(* Logix 5000 project; controller Drives_Line1 1756-L72 rev 20.13; software revision 20.04; part 4 of 21 *)
(* tags used below, declared in another part *)
   EOC_ToCoilerStep : DINT;
   Exit_PosPv_Winder : REAL;
   zMaxSpdExitNotSync : REAL;
   Exit_Accu : UDT_Exit_Accu;
   Exit_PosSp_ToWinder : DINT;
   ExitCmd : UDT_Commands_Zone;
   ExitConfig : UDT_Config_Zone;
   ExitCtrl : UDT_Control_Zone;
   ExitFdbks : UDT_Feedbacks_Zone;
   ExitSetpoints : UDT_Setpoints_Zone;
   ExitStat : UDT_Status_Zone;
   In_Commands : UDT_Commands;
   In_Config : UDT_Config;
   In_Setpoints : UDT_Setpoints;
   LineCmd : UDT_Commands_Line;
   LineStat : UDT_Status_Line;
   Out_Feedbacks : UDT_Fdbks;
   Out_Status : UDT_Status;
   TestConfig_Exit : UDT_Config_Zone;
   Unwinder_1 : UDT_Unwinder;
   Winder : UDT_Winder;
   Winder_FB_Counts_Diff : DINT;
   Winder_FB_Counts_mm : DINT;
   Winder_FB_Update_Valid : BOOL;
   zConfigFromMaster : BOOL;
   zExit_Dist_ShearToWinder : DINT;
   zWinderDiamFullTrq : REAL;
(* P02_Exit_Zone, continued *)

ROUTINE R03_EOC_ToCoiler   (* ladder *)
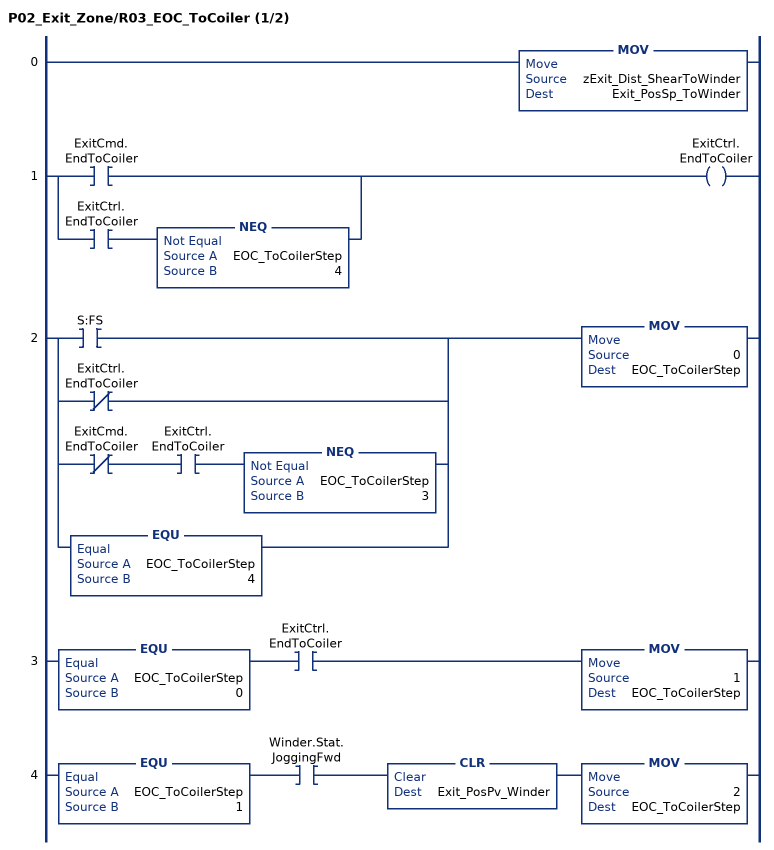
   0: MOV(zExit_Dist_ShearToWinder,Exit_PosSp_ToWinder);
   1: [XIC(ExitCmd.EndToCoiler) ,XIC(ExitCtrl.EndToCoiler) NEQ(EOC_ToCoilerStep,4) ]OTE(ExitCtrl.EndToCoiler);
   2: [XIC(S:FS) ,XIO(ExitCtrl.EndToCoiler) ,XIO(ExitCmd.EndToCoiler) XIC(ExitCtrl.EndToCoiler) NEQ(EOC_ToCoilerStep,3) ,EQU(EOC_ToCoilerStep,4) ]MOV(0,EOC_ToCoilerStep);
   3: EQU(EOC_ToCoilerStep,0)XIC(ExitCtrl.EndToCoiler)MOV(1,EOC_ToCoilerStep);
   4: EQU(EOC_ToCoilerStep,1)XIC(Winder.Stat.JoggingFwd)CLR(Exit_PosPv_Winder)MOV(2,EOC_ToCoilerStep);
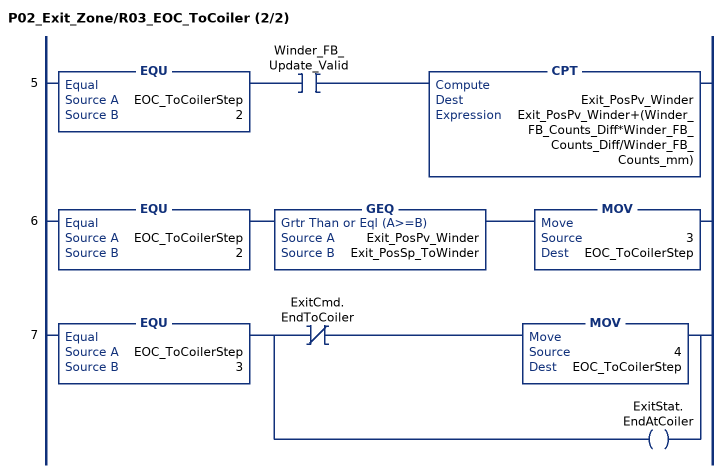
   5: EQU(EOC_ToCoilerStep,2)XIC(Winder_FB_Update_Valid)CPT(Exit_PosPv_Winder,Exit_PosPv_Winder+(Winder_FB_Counts_Diff*Winder_FB_Counts_Diff/Winder_FB_Counts_mm));
   6: EQU(EOC_ToCoilerStep,2)GEQ(Exit_PosPv_Winder,Exit_PosSp_ToWinder)MOV(3,EOC_ToCoilerStep);
   7: EQU(EOC_ToCoilerStep,3)[XIO(ExitCmd.EndToCoiler) MOV(4,EOC_ToCoilerStep) ,OTE(ExitStat.EndAtCoiler) ];
END_ROUTINE

ROUTINE R05_Control   (* ladder *)
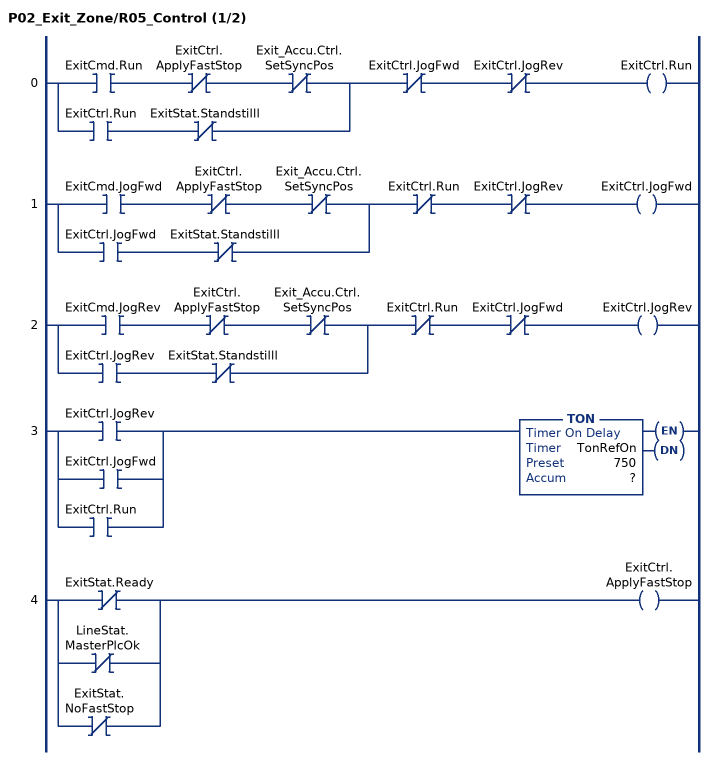
   0: [XIC(ExitCmd.Run) XIO(ExitCtrl.ApplyFastStop) XIO(Exit_Accu.Ctrl.SetSyncPos) ,XIC(ExitCtrl.Run) XIO(ExitStat.Standstilll) ]XIO(ExitCtrl.JogFwd)XIO(ExitCtrl.JogRev)OTE(ExitCtrl.Run);
   1: [XIC(ExitCmd.JogFwd) XIO(ExitCtrl.ApplyFastStop) XIO(Exit_Accu.Ctrl.SetSyncPos) ,XIC(ExitCtrl.JogFwd) XIO(ExitStat.Standstilll) ]XIO(ExitCtrl.Run)XIO(ExitCtrl.JogRev)OTE(ExitCtrl.JogFwd);
   2: [XIC(ExitCmd.JogRev) XIO(ExitCtrl.ApplyFastStop) XIO(Exit_Accu.Ctrl.SetSyncPos) ,XIC(ExitCtrl.JogRev) XIO(ExitStat.Standstilll) ]XIO(ExitCtrl.Run)XIO(ExitCtrl.JogFwd)OTE(ExitCtrl.JogRev);
   3: [XIC(ExitCtrl.JogRev) ,XIC(ExitCtrl.JogFwd) ,XIC(ExitCtrl.Run) ]TON(TonRefOn,?,?);
   4: [XIO(ExitStat.Ready) ,XIO(LineStat.MasterPlcOk) ,XIO(ExitStat.NoFastStop) ]OTE(ExitCtrl.ApplyFastStop);
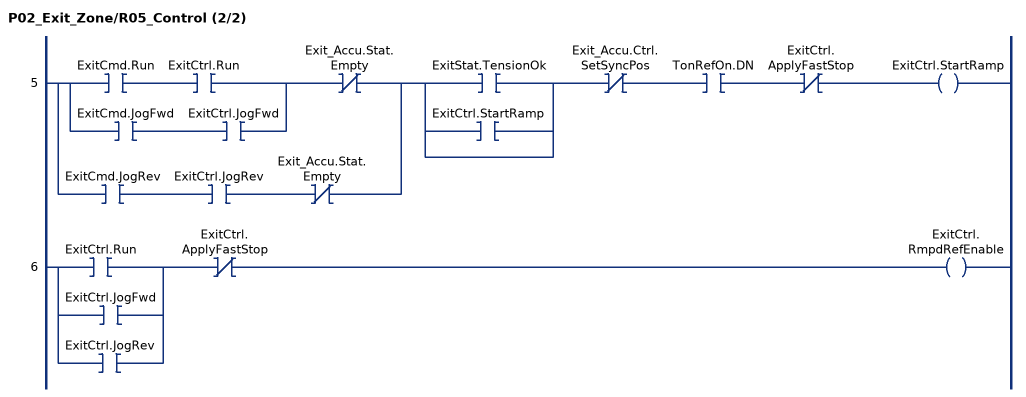
   5: [[XIC(ExitCmd.Run) XIC(ExitCtrl.Run) ,XIC(ExitCmd.JogFwd) XIC(ExitCtrl.JogFwd) ] XIO(Exit_Accu.Stat.Empty) ,XIC(ExitCmd.JogRev) XIC(ExitCtrl.JogRev) XIO(Exit_Accu.Stat.Empty) ][XIC(ExitStat.TensionOk) ,XIC(ExitCtrl.StartRamp) ,]XIO(Exit_Accu.Ctrl.SetSyncPos)XIC(TonRefOn.DN)XIO(ExitCtrl.ApplyFastStop)OTE(ExitCtrl.StartRamp);
   6: [XIC(ExitCtrl.Run) ,XIC(ExitCtrl.JogFwd) ,XIC(ExitCtrl.JogRev) ]XIO(ExitCtrl.ApplyFastStop)OTE(ExitCtrl.RmpdRefEnable);
END_ROUTINE

ROUTINE R07_Ramp_ExitRef_Vx   (* function block diagram *)
   SHEET 1   // Limit speed reference
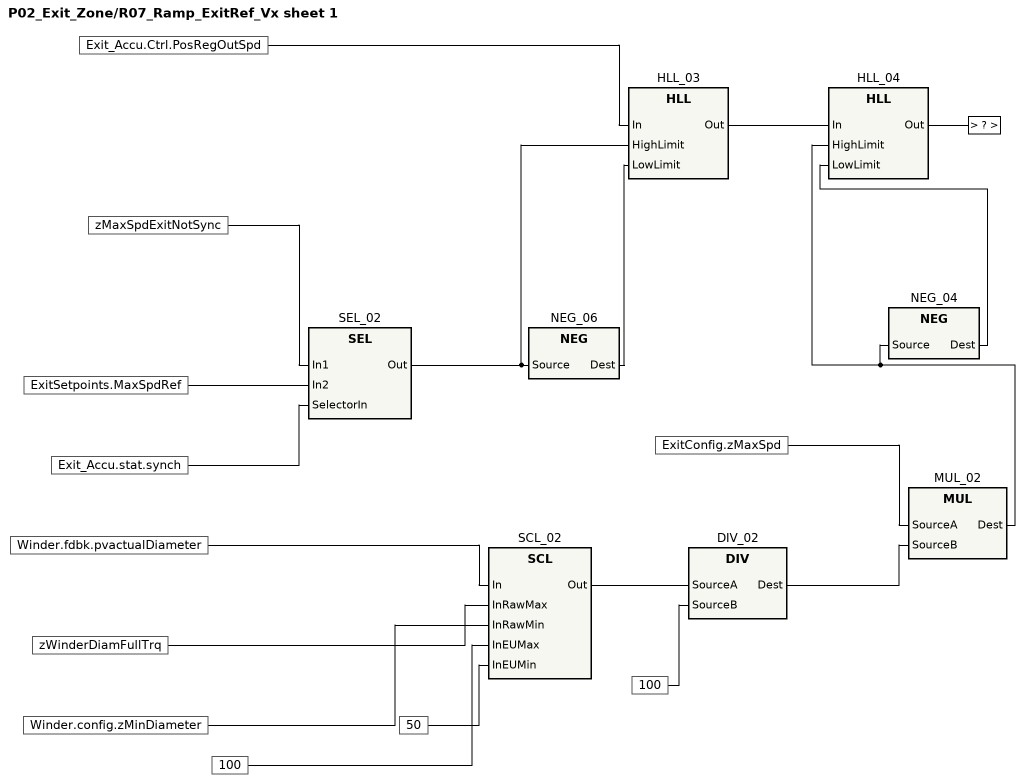
   SEL_02 : SEL(In1 := zMaxSpdExitNotSync, In2 := ExitSetpoints.MaxSpdRef, SelectorIn := Exit_Accu.stat.synch);
   SCL_02 : SCL(In := Winder.fdbk.pvactualDiameter, InRawMax := zWinderDiamFullTrq, InRawMin := Winder.config.zMinDiameter, InEUMax := 100, InEUMin := 50);
   NEG_06 : NEG(Source := SEL_02.Out);
   HLL_03 : HLL(In := Exit_Accu.Ctrl.PosRegOutSpd, HighLimit := SEL_02.Out, LowLimit := NEG_06.Dest);
   DIV_02 : DIV(SourceA := SCL_02.Out, SourceB := 100);
   MUL_02 : MUL(SourceA := ExitConfig.zMaxSpd, SourceB := DIV_02.Dest);
   NEG_04 : NEG(Source := MUL_02.Dest);
   HLL_04 : HLL(In := HLL_03.Out, HighLimit := MUL_02.Dest, LowLimit := NEG_04.Dest);
   WIRE(?) := HLL_04.Out;
   SHEET 2   // Select speed reference
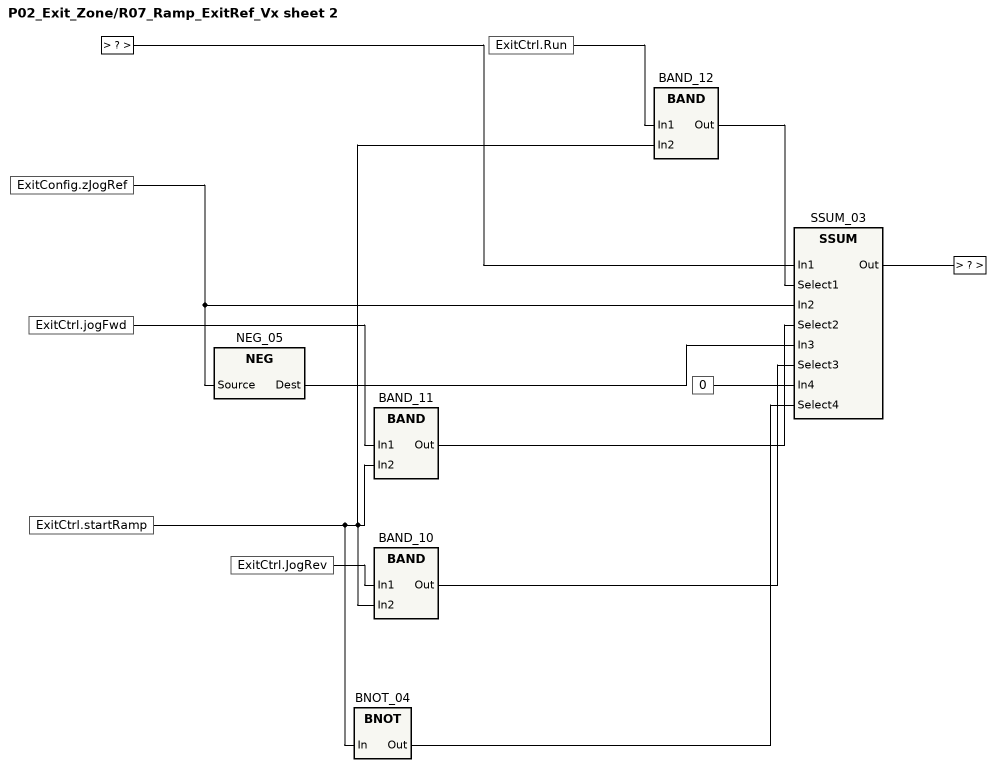
   NEG_05 : NEG(Source := ExitConfig.zJogRef);
   BNOT_04 : BNOT(In := ExitCtrl.startRamp);
   BAND_11 : BAND(In1 := ExitCtrl.jogFwd, In2 := ExitCtrl.startRamp);
   BAND_10 : BAND(In1 := ExitCtrl.JogRev, In2 := ExitCtrl.startRamp);
   BAND_12 : BAND(In1 := ExitCtrl.Run, In2 := ExitCtrl.startRamp);
   SSUM_03 : SSUM(In1 := WIRE(?), Select1 := BAND_12.Out, In2 := ExitConfig.zJogRef, Select2 := BAND_11.Out, In3 := NEG_05.Dest, Select3 := BAND_10.Out, In4 := 0, Select4 := BNOT_04.Out);
   WIRE(?) := SSUM_03.Out;
   SHEET 3   // Select acceleration rate
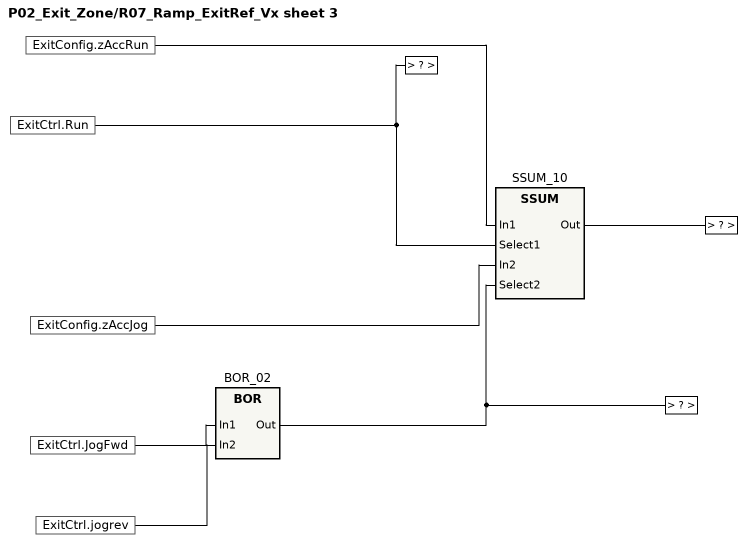
   BOR_02 : BOR(In1 := ExitCtrl.JogFwd, In2 := ExitCtrl.jogrev);
   WIRE(?) := ExitCtrl.Run;
   SSUM_10 : SSUM(In1 := ExitConfig.zAccRun, Select1 := ExitCtrl.Run, In2 := ExitConfig.zAccJog, Select2 := BOR_02.Out);
   WIRE(?) := BOR_02.Out;
   WIRE(?) := SSUM_10.Out;
   SHEET 4   // Select deceleration rate
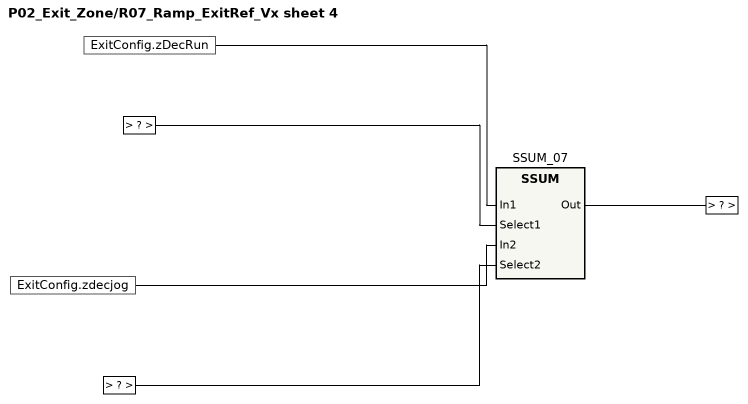
   SSUM_07 : SSUM(In1 := ExitConfig.zDecRun, Select1 := WIRE(?), In2 := ExitConfig.zdecjog, Select2 := WIRE(?));
   WIRE(?) := SSUM_07.Out;
   SHEET 5   // Select jerk rate
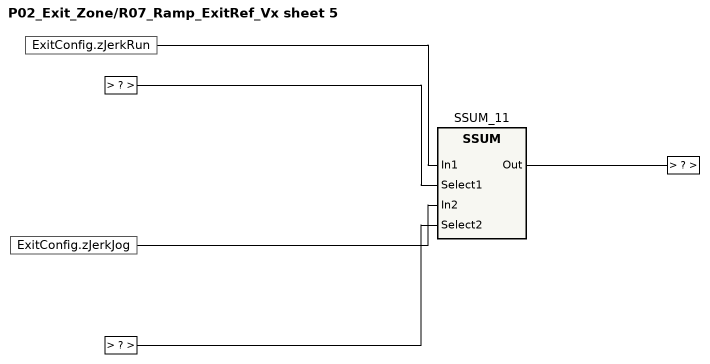
   SSUM_11 : SSUM(In1 := ExitConfig.zJerkRun, Select1 := WIRE(?), In2 := ExitConfig.zJerkJog, Select2 := WIRE(?));
   WIRE(?) := SSUM_11.Out;
   SHEET 6   // S-Curve entry speed (Ve)
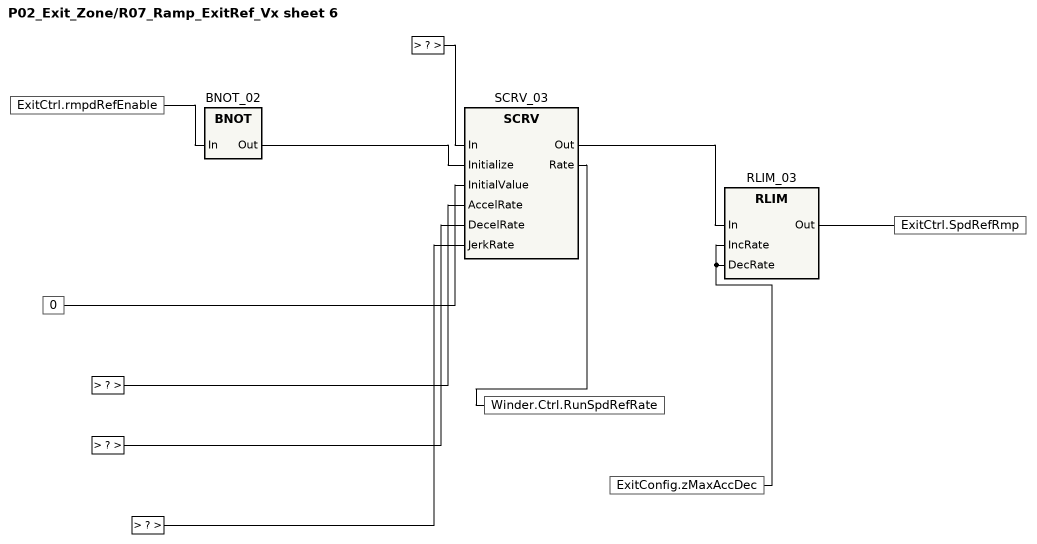
   BNOT_02 : BNOT(In := ExitCtrl.rmpdRefEnable);
   SCRV_03 : SCRV(In := WIRE(?), Initialize := BNOT_02.Out, InitialValue := 0, AccelRate := WIRE(?), DecelRate := WIRE(?), JerkRate := WIRE(?));
   Winder.Ctrl.RunSpdRefRate := SCRV_03.Rate;
   RLIM_03 : RLIM(In := SCRV_03.Out, IncRate := ExitConfig.zMaxAccDec, DecRate := ExitConfig.zMaxAccDec);
   ExitCtrl.SpdRefRmp := RLIM_03.Out;
END_ROUTINE

ROUTINE R999_Test   (* ladder *)
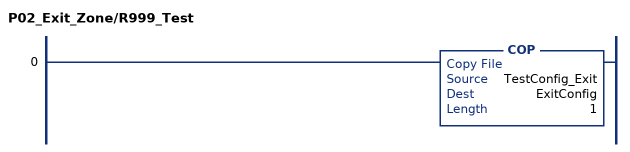
   0: COP(TestConfig_Exit,ExitConfig,1);
END_ROUTINE

ROUTINE R99_To_Master   (* ladder *)
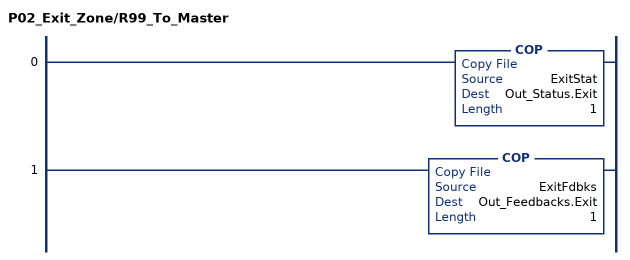
   0: COP(ExitStat,Out_Status.Exit,1);
   1: COP(ExitFdbks,Out_Feedbacks.Exit,1);
END_ROUTINE
END_PROGRAM

PROGRAM P10_Unwinder_1   (* main routine R00_Main *)
VAR
   ABS_01 : FBD_MATH_ADVANCED; {access Read Only}
   ABS_02 : FBD_MATH_ADVANCED;
   ABS_03 : FBD_MATH_ADVANCED;
   ABS_04 : FBD_MATH_ADVANCED;
   ADD_03 : FBD_MATH;
   BAND_01 : FBD_BOOLEAN_AND := (In3 := 1, In4 := 1, In5 := 1, In6 := 1, In7 := 1, In8 := 1);
   BAND_02 : FBD_BOOLEAN_AND := (In4 := 1, In5 := 1, In6 := 1, In7 := 1, In8 := 1);
   BAND_03 : FBD_BOOLEAN_AND := (In3 := 1, In4 := 1, In5 := 1, In6 := 1, In7 := 1, In8 := 1);
   BAND_04 : FBD_BOOLEAN_AND := (In3 := 1, In4 := 1, In5 := 1, In6 := 1, In7 := 1, In8 := 1);
   BAND_05 : FBD_BOOLEAN_AND := (In3 := 1, In4 := 1, In5 := 1, In6 := 1, In7 := 1, In8 := 1);
   BAND_06 : FBD_BOOLEAN_AND := (In1 := 1, In3 := 1, In4 := 1, In5 := 1, In6 := 1, In7 := 1, In8 := 1);
   BAND_07 : FBD_BOOLEAN_AND := (In3 := 1, In4 := 1, In5 := 1, In6 := 1, In7 := 1, In8 := 1);
   BAND_08 : FBD_BOOLEAN_AND := (In3 := 1, In4 := 1, In5 := 1, In6 := 1, In7 := 1, In8 := 1);
   BAND_11 : FBD_BOOLEAN_AND := (In3 := 1, In4 := 1, In5 := 1, In6 := 1, In7 := 1, In8 := 1);
   BNOT_01 : FBD_BOOLEAN_NOT := (Out := 1);
   BNOT_02 : FBD_BOOLEAN_NOT := (Out := 1);
   BNOT_04 : FBD_BOOLEAN_NOT := (Out := 1);
   BNOT_06 : FBD_BOOLEAN_NOT := (Out := 1);
   BNOT_07 : FBD_BOOLEAN_NOT := (Out := 1);
   BNOT_08 : FBD_BOOLEAN_NOT := (Out := 1);
   BOR_01 : FBD_BOOLEAN_OR := (In1 := 1, Out := 1);
   BOR_03 : FBD_BOOLEAN_OR;
   BOR_04 : FBD_BOOLEAN_OR;
   Diamtest : BOOL;
   Diamtest_mm : REAL := 1080.0;
   DIV_01 : FBD_MATH := (SourceA := 2.5, SourceB := 100.0, Dest := 0.025);
   DIV_02 : FBD_MATH := (SourceB := 78.0);
   DIV_04 : FBD_MATH := (SourceB := 1440.0);
   DIV_10 : FBD_MATH := (Dest := 2498.0051);
   DIV_11 : FBD_MATH := (SourceA := 2498.0051, SourceB := 3.1415927, Dest := 795.1397);
   DIV_12 : FBD_MATH := (SourceB := 60.0);
   DIV_14 : FBD_MATH := (SourceB := 0.0048139803);
   DIV_15 : FBD_MATH := (SourceA := 100.0, SourceB := 100.0, Dest := 1.0);
   EQU_01 : FBD_COMPARE := (SourceA := 1.0, SourceB := 4.0);
   FGEN_01 : FUNCTION_GENERATOR := (XY1Size := 21);
   GEQ_02 : FBD_COMPARE := (SourceB := 0.5);
   GRT_01 : FBD_COMPARE := (SourceB := 1.e-04);
   HLL_01 : HL_LIMIT := (In := 547.79364, HighLimit := 2000.0, LowLimit := 500.0, Out := 547.79364);
   HLL_07 : HL_LIMIT := (In := 9950.0, HighLimit := 15000.0, Out := 9950.0);
   INTG_01 : INTEGRATOR := (Initialize := 1, IGain := 1000.02, RTSTime := 1, DeltaT := 0.05);
   INTG_02 : INTEGRATOR := (Initialize := 1, IGain := 0.016666, RTSTime := 1, DeltaT := 0.05);
   IO_State_Tmp_Unwinder_1 : INT := 16384;
   IO_State_Unwinder_1 : INT := 4;
   LES_01 : FBD_COMPARE;
   LPF_02 : FILTER_LOW_PASS := (WLag := 10.0, Order := 1, RTSTime := 1, DeltaT := 0.05); {access Read Only}
   LPF_1000 : FILTER_LOW_PASS := (WLag := 10.0, Order := 1, RTSTime := 1, DeltaT := 0.05);
   LPF_1006 : FILTER_LOW_PASS := (WLag := 10.0, Order := 1, RTSTime := 1, DeltaT := 0.05);
   MUL_01 : FBD_MATH := (SourceB := 2719.4368);
   MUL_02 : FBD_MATH := (SourceB := 0.0048139803);
   MUL_03 : FBD_MATH := (SourceB := 25.0);
   MUL_04 : FBD_MATH := (SourceB := 100.0);
   MUL_05 : FBD_MATH := (SourceB := 0.5);
   MUL_06 : FBD_MATH := (SourceA := 0.5, SourceB := 5.0, Dest := 2.5);
   MUL_07 : FBD_MATH := (SourceA := 1.0057888);
   MUL_23 : FBD_MATH := (SourceA := 9950.0, SourceB := 1.0, Dest := 9950.0);
   MUL_26 : FBD_MATH := (SourceB := 2719.4368);
   NEG_01 : FBD_MATH_ADVANCED := (Source := 0.083, Dest := -0.083);
   NEG_02 : FBD_MATH_ADVANCED;
   NEG_03 : FBD_MATH_ADVANCED;
   NEG_04 : FBD_MATH_ADVANCED;
   RLIM_01 : RATE_LIMITER := (In := 795.1397, RTSTime := 1, Out := 547.79364, DeltaT := 0.05);
   RLIM_03 : RATE_LIMITER := (IncRate := 0.25, DecRate := 0.25, RTSTime := 1, DeltaT := 0.05);
   RLIM_04 : RATE_LIMITER := (IncRate := 5000.0, DecRate := 5000.0, ByPass := 1, RTSTime := 1, DeltaT := 0.05);
   SCL_01 : SCALE := (In := 512.2091, InRawMax := 5851.2163, InEUMax := 35.0, InEUMin := 25.0, Limiting := 1, Out := 25.87539);
   SCL_02 : SCALE := (InRawMax := 0.5, InEUMax := 10.0, InEUMin := 5.0, Limiting := 1, Out := 5.0);
   SCRV_02 : S_CURVE := (Initialize := 1, AbsAlgRamp := 1, AccelRate := 0.16, DecelRate := 0.16, JerkRate := 0.25, RTSTime := 1, DeltaT := 0.05);
   SEL_01 : SELECT;
   SEL_02 : SELECT := (In2 := 0.025);
   SEL_03 : SELECT;
   SEL_04 : SELECT;
   SEL_05 : SELECT := (In1 := 795.1397, In2 := 800.0, Out := 795.1397);
   SEL_06 : SELECT := (In1 := 547.79364, In2 := 1080.0, Out := 547.79364);
   SEL_07 : SELECT := (In1 := 0.5, In2 := 0.5, Out := 0.5);
   SEL_08 : SELECT := (In1 := 795.1397, In2 := 800.0, Out := 795.1397);
   SEL_18 : SELECT := (In1 := 9950.0, SelectorIn := 1);
   SSUM_01 : SELECTED_SUMMER := (In1 := 9950.0, Gain1 := 1.0, Select1 := 1, In2 := 9950.0, Gain2 := 1.0, Gain3 := 1.0, Gain4 := 1.0, Gain5 := 1.0, Gain6 := 1.0, Gain7 := 1.0, Gain8 := 1.0, Out := 9950.0);
   SSUM_02 : SELECTED_SUMMER := (In1 := 0.083, Gain1 := 1.0, In2 := -0.083, Gain2 := 1.0, Gain3 := 1.0, Select3 := 1, Gain4 := 1.0, Gain5 := 1.0, Gain6 := 1.0, Gain7 := 1.0, Gain8 := 1.0);
   SSUM_03 : SELECTED_SUMMER := (Gain1 := 1.0, Select1 := 1, Gain2 := 1.0, Gain3 := 1.0, Gain4 := 1.0, Gain5 := 1.0, Gain6 := 1.0, Gain7 := 1.0, Gain8 := 1.0);
   SSUM_04 : SELECTED_SUMMER := (Gain1 := 1.0, Select1 := 1, Gain2 := 1.0, Gain3 := 1.0, Gain4 := 1.0, Gain5 := 1.0, Gain6 := 1.0, Gain7 := 1.0, Gain8 := 1.0);
   SSUM_05 : SELECTED_SUMMER := (Gain1 := 1.0, Gain2 := 1.0, Gain3 := 1.0, Gain4 := 1.0, Gain5 := 1.0, Gain6 := 1.0, Gain7 := 1.0, Gain8 := 1.0);
   SUB_08 : FBD_MATH; {access Read Only}
   TimeForBr : TIMER := (PRE := 750);
   TimeOffBr : TIMER := (PRE := 2000, ACC := 2000);
   TimeOffFan : TIMER := (PRE := 180000, ACC := 180049);
   TofReset : TIMER := (PRE := 1000, ACC := 1000);
   TonNoResponse : TIMER := (PRE := 2500);
   TonRefOn : TIMER := (PRE := 750);
   TonTensionOnSp : TIMER := (PRE := 1000);
   Unwinder_1_DiamCalcOn : BOOL;
   Unwinder_1_JEC : REAL := 1.0; {access Read Only}
   Unwinder_1_JLossCrvSpd : REAL[21] := ([0] := -1500.0, [1] := -1350.0, [2] := -1200.0, [3] := -1050.0, [4] := -900.0, [5] := -750.0, [6] := -600.0, [7] := -450.0, [8] := -300.0, [9] := -150.0, [11] := 150.0, [12] := 300.0, [13] := 450.0, [14] := 600.0, [15] := 750.0, [16] := 900.0, [17] := 1050.0, [18] := 1200.0, [19] := 1350.0, [20] := 1500.0);
   Unwinder_1_JMaterial : REAL := 0.0057888483; {access Read Only}
   Unwinder_1_LossCrvTrq_Pct : REAL[21] := ([0] := -6.5, [1] := -6.5, [2] := -6.5, [3] := -6.5, [4] := -6.5, [5] := -6.5, [6] := -6.0, [7] := -6.0, [8] := -5.0, [9] := -3.9, [11] := 3.9, [12] := 6.2, [13] := 7.0, [14] := 7.5, [15] := 7.5, [16] := 7.5, [17] := 7.5, [18] := 7.5, [19] := 7.5, [20] := 7.5);
   Unwinder_1_MatMass : REAL := 512.2091; {access Read Only}
   Unwinder_1_MatVolume : REAL := 0.1375058; {access Read Only}
   Unwinder_1_MaxMass : REAL := 5851.2163;
   Unwinder_1_MaxVolume : REAL := 1.5707964;
   Unwinder_1_PctPerN : REAL := 0.0048139803; {access Read Only}
   Unwinder_1_RatedTrq : REAL := 72.94375; {access Read Only}
   Unwinder_1_RPMPerMPS : REAL := 2719.4368;
   Unwinder_1_Running : BOOL;
   Unwinder_1_SpdMps_Flt : REAL;
   Unwinder_1_SpdRpm_Flt : REAL;
   zUnwinder_1_JGainQ1Q2 : REAL := 0.5;
   zUnwinder_1_JGainQ3Q4 : REAL := 0.5;
   zUnwinder_1_RateMax : REAL := 0.25;
   zUnwinder_1_SpdReg_BWMax : REAL := 35.0;
   zUnwinder_1_SpdReg_BWmin : REAL := 25.0;
   zUnwinder_1_Stall_Spd : REAL := 10.0;
   zUnwinder_1_TenRefRate : REAL := 5000.0;
   zUnwinder_1_Tens_Offs : REAL := 25.0;
   zUnwinder_1_TenSpStall : REAL := 100.0;
   zUnwinder_1_TrqTrimLimMax_Pct : REAL := 10.0;
   zUnwinder_1_TrqTrimLimMin_Pct : REAL := 5.0;
END_VAR

ROUTINE R00_Main   (* ladder *)
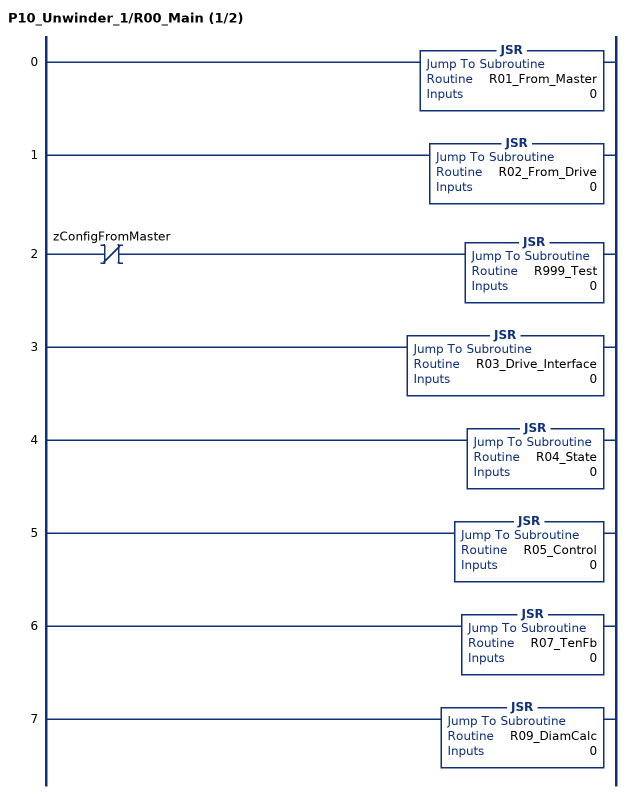
   0: JSR(R01_From_Master,0);
   1: JSR(R02_From_Drive,0);
   2: XIO(zConfigFromMaster)JSR(R999_Test,0);
   3: JSR(R03_Drive_Interface,0);
   4: JSR(R04_State,0);
   5: JSR(R05_Control,0);
   6: JSR(R07_TenFb,0);
   7: JSR(R09_DiamCalc,0);
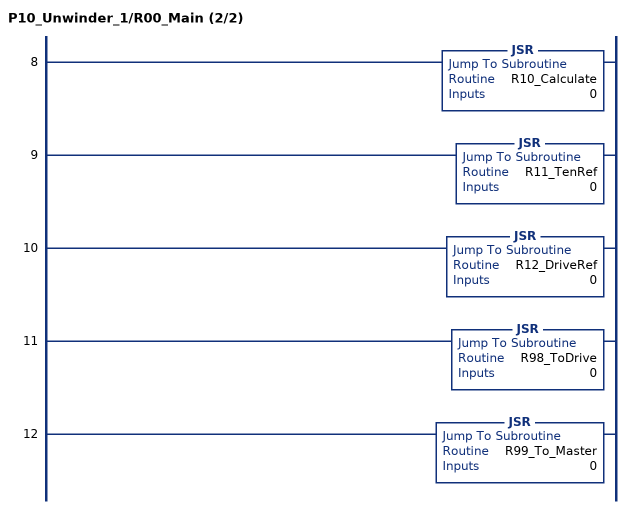
   8: JSR(R10_Calculate,0);
   9: JSR(R11_TenRef,0);
   10: JSR(R12_DriveRef,0);
   11: JSR(R98_ToDrive,0);
   12: JSR(R99_To_Master,0);
END_ROUTINE

ROUTINE R01_From_Master   (* ladder *)
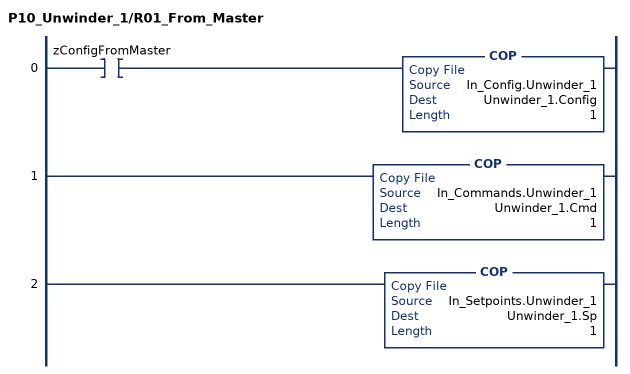
   0: XIC(zConfigFromMaster)COP(In_Config.Unwinder_1,Unwinder_1.Config,1);
   1: COP(In_Commands.Unwinder_1,Unwinder_1.Cmd,1);
   2: COP(In_Setpoints.Unwinder_1,Unwinder_1.Sp,1);
END_ROUTINE

ROUTINE R02_From_Drive   (* ladder *)
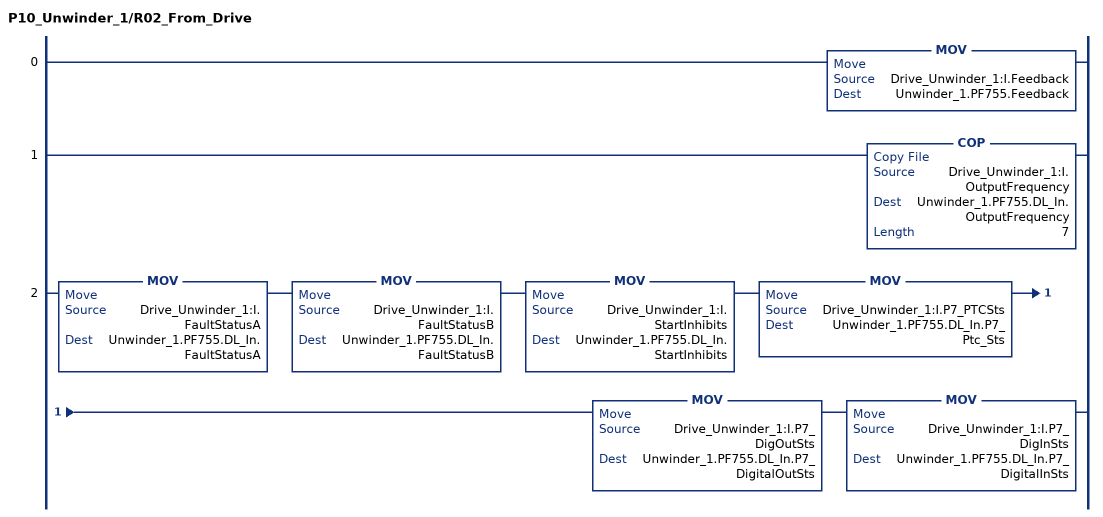
   0: MOV(Drive_Unwinder_1:I.Feedback,Unwinder_1.PF755.Feedback);
   1: COP(Drive_Unwinder_1:I.OutputFrequency,Unwinder_1.PF755.DL_In.OutputFrequency,7);
   2: MOV(Drive_Unwinder_1:I.FaultStatusA,Unwinder_1.PF755.DL_In.FaultStatusA)MOV(Drive_Unwinder_1:I.FaultStatusB,Unwinder_1.PF755.DL_In.FaultStatusB)MOV(Drive_Unwinder_1:I.StartInhibits,Unwinder_1.PF755.DL_In.StartInhibits)MOV(Drive_Unwinder_1:I.P7_PTCSts,Unwinder_1.PF755.DL_In.P7_Ptc_Sts)MOV(Drive_Unwinder_1:I.P7_DigOutSts,Unwinder_1.PF755.DL_In.P7_DigitalOutSts)MOV(Drive_Unwinder_1:I.P7_DigInSts,Unwinder_1.PF755.DL_In.P7_DigitalInSts);
END_ROUTINE

ROUTINE R03_Drive_Interface   (* ladder *)
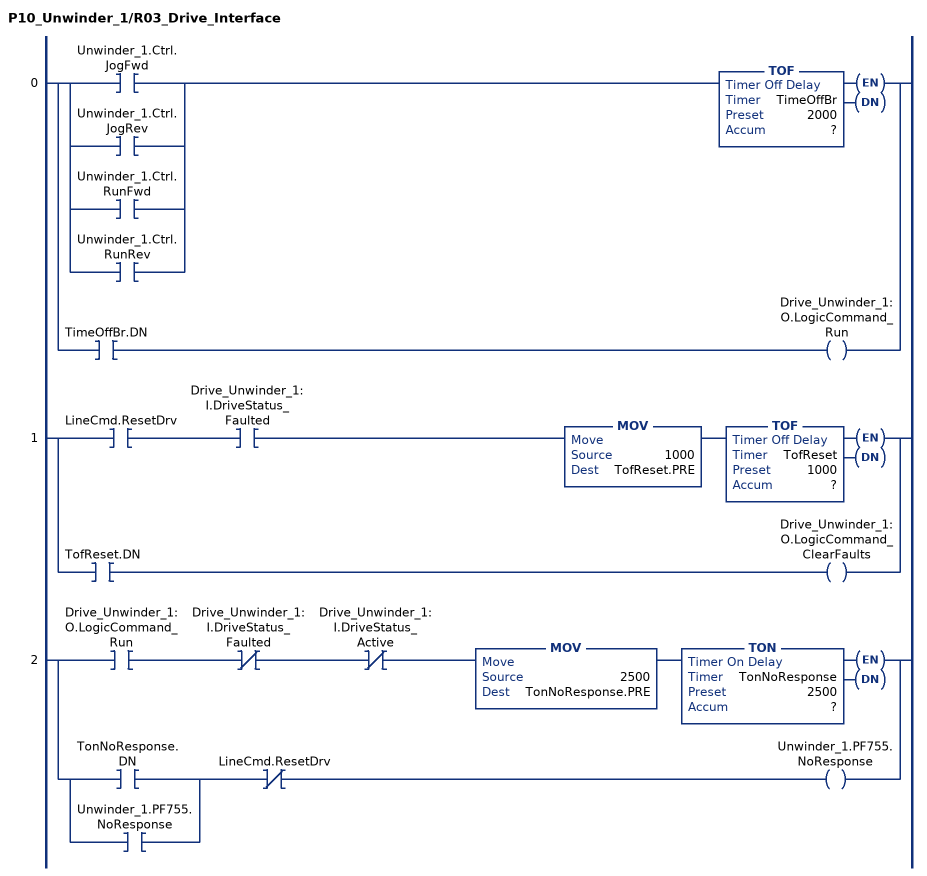
   0: [[XIC(Unwinder_1.Ctrl.JogFwd) ,XIC(Unwinder_1.Ctrl.JogRev) ,XIC(Unwinder_1.Ctrl.RunFwd) ,XIC(Unwinder_1.Ctrl.RunRev) ] TOF(TimeOffBr,?,?) ,XIC(TimeOffBr.DN) OTE(Drive_Unwinder_1:O.LogicCommand_Run) ];
   1: [XIC(LineCmd.ResetDrv) XIC(Drive_Unwinder_1:I.DriveStatus_Faulted) MOV(1000,TofReset.PRE) TOF(TofReset,?,?) ,XIC(TofReset.DN) OTE(Drive_Unwinder_1:O.LogicCommand_ClearFaults) ];
   2: [XIC(Drive_Unwinder_1:O.LogicCommand_Run) XIO(Drive_Unwinder_1:I.DriveStatus_Faulted) XIO(Drive_Unwinder_1:I.DriveStatus_Active) MOV(2500,TonNoResponse.PRE) TON(TonNoResponse,?,?) ,[XIC(TonNoResponse.DN) ,XIC(Unwinder_1.PF755.NoResponse) ] XIO(LineCmd.ResetDrv) OTE(Unwinder_1.PF755.NoResponse) ];
END_ROUTINE

ROUTINE R04_State   (* ladder *)
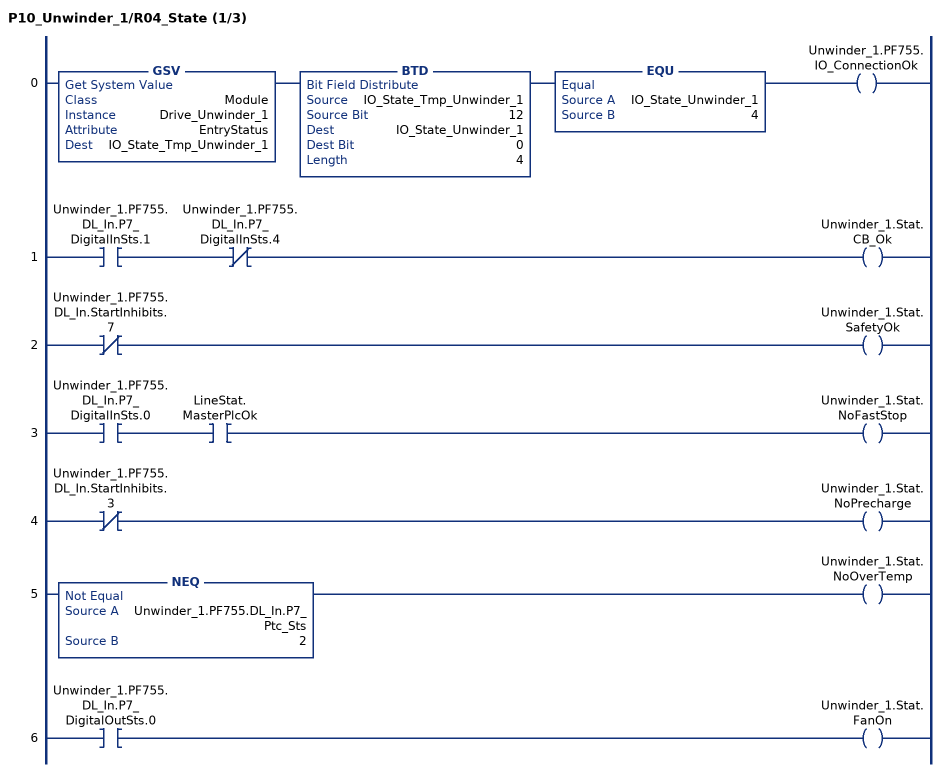
   0: GSV(Module,Drive_Unwinder_1,EntryStatus,IO_State_Tmp_Unwinder_1)BTD(IO_State_Tmp_Unwinder_1,12,IO_State_Unwinder_1,0,4)EQU(IO_State_Unwinder_1,4)OTE(Unwinder_1.PF755.IO_ConnectionOk);
   1: XIC(Unwinder_1.PF755.DL_In.P7_DigitalInSts.1)XIO(Unwinder_1.PF755.DL_In.P7_DigitalInSts.4)OTE(Unwinder_1.Stat.CB_Ok);
   2: XIO(Unwinder_1.PF755.DL_In.StartInhibits.7)OTE(Unwinder_1.Stat.SafetyOk);
   3: XIC(Unwinder_1.PF755.DL_In.P7_DigitalInSts.0)XIC(LineStat.MasterPlcOk)OTE(Unwinder_1.Stat.NoFastStop);
   4: XIO(Unwinder_1.PF755.DL_In.StartInhibits.3)OTE(Unwinder_1.Stat.NoPrecharge);
   5: NEQ(Unwinder_1.PF755.DL_In.P7_Ptc_Sts,2)OTE(Unwinder_1.Stat.NoOverTemp);
   6: XIC(Unwinder_1.PF755.DL_In.P7_DigitalOutSts.0)OTE(Unwinder_1.Stat.FanOn);
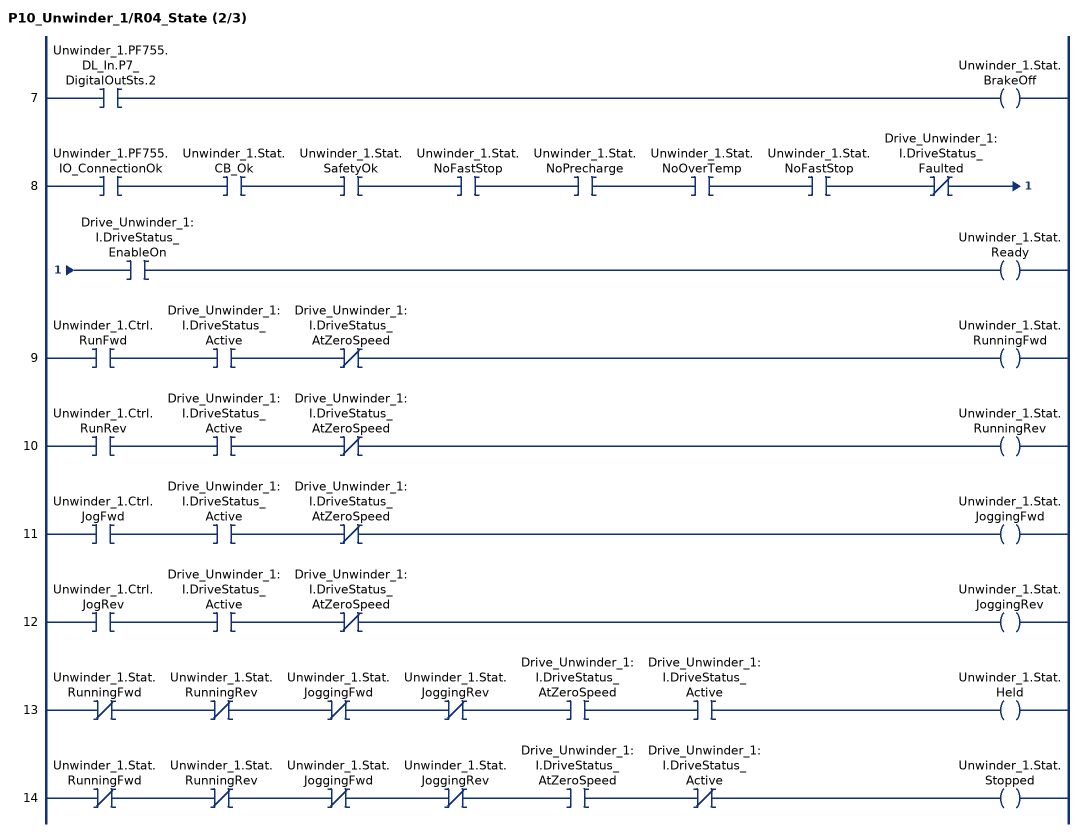
   7: XIC(Unwinder_1.PF755.DL_In.P7_DigitalOutSts.2)OTE(Unwinder_1.Stat.BrakeOff);
   8: XIC(Unwinder_1.PF755.IO_ConnectionOk)XIC(Unwinder_1.Stat.CB_Ok)XIC(Unwinder_1.Stat.SafetyOk)XIC(Unwinder_1.Stat.NoFastStop)XIC(Unwinder_1.Stat.NoPrecharge)XIC(Unwinder_1.Stat.NoOverTemp)XIC(Unwinder_1.Stat.NoFastStop)XIO(Drive_Unwinder_1:I.DriveStatus_Faulted)XIC(Drive_Unwinder_1:I.DriveStatus_EnableOn)OTE(Unwinder_1.Stat.Ready);
   9: XIC(Unwinder_1.Ctrl.RunFwd)XIC(Drive_Unwinder_1:I.DriveStatus_Active)XIO(Drive_Unwinder_1:I.DriveStatus_AtZeroSpeed)OTE(Unwinder_1.Stat.RunningFwd);
   10: XIC(Unwinder_1.Ctrl.RunRev)XIC(Drive_Unwinder_1:I.DriveStatus_Active)XIO(Drive_Unwinder_1:I.DriveStatus_AtZeroSpeed)OTE(Unwinder_1.Stat.RunningRev);
   11: XIC(Unwinder_1.Ctrl.JogFwd)XIC(Drive_Unwinder_1:I.DriveStatus_Active)XIO(Drive_Unwinder_1:I.DriveStatus_AtZeroSpeed)OTE(Unwinder_1.Stat.JoggingFwd);
   12: XIC(Unwinder_1.Ctrl.JogRev)XIC(Drive_Unwinder_1:I.DriveStatus_Active)XIO(Drive_Unwinder_1:I.DriveStatus_AtZeroSpeed)OTE(Unwinder_1.Stat.JoggingRev);
   13: XIO(Unwinder_1.Stat.RunningFwd)XIO(Unwinder_1.Stat.RunningRev)XIO(Unwinder_1.Stat.JoggingFwd)XIO(Unwinder_1.Stat.JoggingRev)XIC(Drive_Unwinder_1:I.DriveStatus_AtZeroSpeed)XIC(Drive_Unwinder_1:I.DriveStatus_Active)OTE(Unwinder_1.Stat.Held);
   14: XIO(Unwinder_1.Stat.RunningFwd)XIO(Unwinder_1.Stat.RunningRev)XIO(Unwinder_1.Stat.JoggingFwd)XIO(Unwinder_1.Stat.JoggingRev)XIC(Drive_Unwinder_1:I.DriveStatus_AtZeroSpeed)XIO(Drive_Unwinder_1:I.DriveStatus_Active)OTE(Unwinder_1.Stat.Stopped);
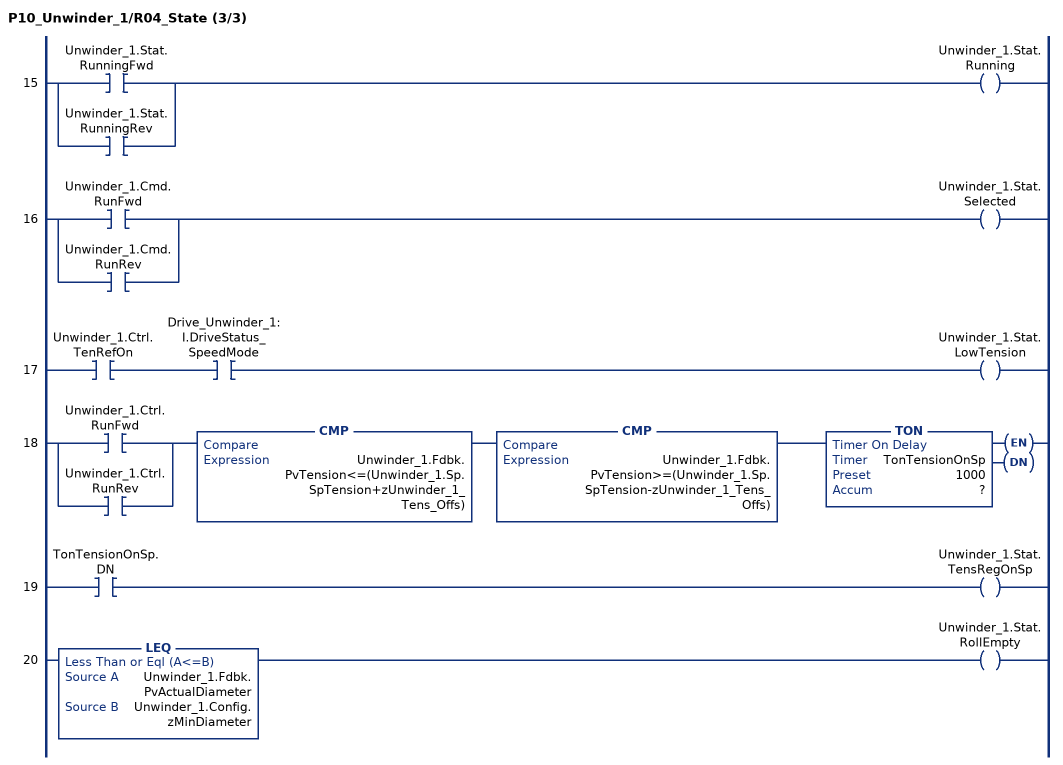
   15: [XIC(Unwinder_1.Stat.RunningFwd) ,XIC(Unwinder_1.Stat.RunningRev) ]OTE(Unwinder_1.Stat.Running);
   16: [XIC(Unwinder_1.Cmd.RunFwd) ,XIC(Unwinder_1.Cmd.RunRev) ]OTE(Unwinder_1.Stat.Selected);
   17: XIC(Unwinder_1.Ctrl.TenRefOn)XIC(Drive_Unwinder_1:I.DriveStatus_SpeedMode)OTE(Unwinder_1.Stat.LowTension);
   18: [XIC(Unwinder_1.Ctrl.RunFwd) ,XIC(Unwinder_1.Ctrl.RunRev) ]CMP(Unwinder_1.Fdbk.PvTension<=(Unwinder_1.Sp.SpTension+zUnwinder_1_Tens_Offs))CMP(Unwinder_1.Fdbk.PvTension>=(Unwinder_1.Sp.SpTension-zUnwinder_1_Tens_Offs))TON(TonTensionOnSp,?,?);
   19: XIC(TonTensionOnSp.DN)OTE(Unwinder_1.Stat.TensRegOnSp);
   20: LEQ(Unwinder_1.Fdbk.PvActualDiameter,Unwinder_1.Config.zMinDiameter)OTE(Unwinder_1.Stat.RollEmpty);
END_ROUTINE
